(* states according to PackTags v3.0 *)
//==================================================================================================
//								RJM Maszyny sp. z o.o.
//									27.06.2022
//	Spis dostepnych stanow maszyny
// 	v1.0	|| TC v 3.1.4024.29		|| - pierwsza wersja
//==================================================================================================
{attribute 'qualified_only'}
{attribute 'strict'}
TYPE E_PMLState :
(
	UNDEFINED		:=  0,
	CLEARING 		:=  1,
	STOPPED 		:=  2,
	STARTING 		:=  3,
	IDLE 			:=  4,
	SUSPENDED 		:=  5,
	EXECUTE 		:=  6,
	STOPPING	 	:=  7,
	ABORTING 		:=  8,
	ABORTED 		:=  9,
	HOLDING 		:= 10,
	HELD 			:= 11,
	UNHOLDING 		:= 12,
	SUSPENDING 		:= 13,
	UNSUSPENDING 	:= 14,
	RESETTING 		:= 15,
	COMPLETING 		:= 16,
	COMPLETE	 	:= 17
);
END_TYPE

(* stored: Version 1.1.0.1, ProductVersion 3.1.4024.11
   DUT E_PMLState: Id {b5dd7f12-0401-4f5d-87ae-a29ba4f07432} *)
